// TIA Portal V20 export
DATA_BLOCK "Stations"   // DB11
{ S7_Optimized_Access := 'TRUE' }
// stored: MemoryReserve 100
   VAR
      ST31_FL1 : "Station";
      ST31_FL2 { S7_SetPoint := 'True'} : "Station";
      ST31_FL3 { S7_SetPoint := 'True'} : "Station";
      ST31_FL4 { S7_SetPoint := 'True'} : "Station";
      ST31_FL5 { S7_SetPoint := 'True'} : "Station";
      ST31_FL6 { S7_SetPoint := 'True'} : "Station";
      ST32_FL1 : "Station";
      ST32_FL2 { S7_SetPoint := 'True'} : "Station";
      ST32_FL3 { S7_SetPoint := 'True'} : "Station";
      ST32_FL4 { S7_SetPoint := 'True'} : "Station";
      ST32_FL5 { S7_SetPoint := 'True'} : "Station";
      ST32_FL6 { S7_SetPoint := 'True'} : "Station";
      ST34_FL1 : "Station";
      ST34_FL2 { S7_SetPoint := 'True'} : "Station";
      ST34_FL3 { S7_SetPoint := 'True'} : "Station";
      ST34_FL4 { S7_SetPoint := 'True'} : "Station";
      ST34_FL5 { S7_SetPoint := 'True'} : "Station";
      ST34_FL6 { S7_SetPoint := 'True'} : "Station";
   END_VAR
BEGIN
END_DATA_BLOCK
